FUNCTION BOOL_TO_QUARTER
  (* Standard: 61499-1; Description: Copyright (c) 2024 HR Agrartechnik GmbH This program and the accompanying materials are made available under the terms of the Eclipse Public License 2.0 which is available at https://www.eclipse.org/legal/epl-2.0/ SPDX-License-Identifier: EPL-2.0 *)
  (* Version 1.0, 2024-02-29, Franz Höpfinger, HR Agrartechnik GmbH *)
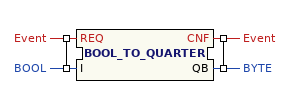
  EVENT_INPUT
    REQ WITH I;
  END_EVENT
  EVENT_OUTPUT
    CNF WITH QB;
  END_EVENT
  VAR_INPUT
    I : BOOL := BOOL#FALSE; (* BOOL Input *)
  END_VAR
  VAR_OUTPUT
    QB : BYTE := COMMAND_DISABLE; (* 2bit (quarter Byte) Output with 4 States (only 2 used) *)
  END_VAR
  BODY IN ST:
FUNCTION BOOL_TO_QUARTER

VAR_INPUT
	I : BOOL := BOOL#FALSE;    // BOOL Input
END_VAR

VAR_OUTPUT
	QB : BYTE := COMMAND_DISABLE;    // 2bit (quarter Byte) Output with 4 States (only 2 used)
END_VAR

CASE I OF
	BOOL#TRUE :
		QB := COMMAND_ENABLE;
	ELSE
		QB := COMMAND_DISABLE;
END_CASE;

END_FUNCTION
  END_BODY
END_FUNCTION
